TYPE Pieza:
STRUCT
    TipoPieza : CaracteristicasPieza;		
	BienColocada    : BOOL := FALSE;
	EsBuena : BOOL := FALSE;
END_STRUCT
END_TYPE

(* stored: Version 1.1.0.1, ProductVersion 3.1.4024.12
   DUT Pieza: Id {791fa912-3ef6-4d8f-811e-2b149a22260a} *)
